Fanuc TP program (LS listing): DEP_CONDMON.LS

/PROG  DEP_CONDMON	  Cond
/ATTR
OWNER		= MNEDITOR;
COMMENT		= "";
PROG_SIZE	= 174;
CREATE		= DATE 25-01-23  TIME 17:34:20;
MODIFIED	= DATE 25-02-06  TIME 18:19:30;
FILE_NAME	= ;
VERSION		= 0;
LINE_COUNT	= 1;
MEMORY_SIZE	= 550;
PROTECT		= READ_WRITE;
TCD:  STACK_SIZE	= 0,
      TASK_PRIORITY	= 50,
      TIME_SLICE	= 0,
      BUSY_LAMP_OFF	= 0,
      ABORT_REQUEST	= 0,
      PAUSE_REQUEST	= 0;
DEFAULT_GROUP	= *,*,*,*,*;
CONTROL_CODE	= 00000000 00000000;
/APPL
/MN
   1:  WHEN GI[47]<50 OR GI[48]<50,CALL DEP_ACTPROG ;
/POS
/END
